(* IEC 61131-3 sources: Modbus-TCP-Traffic-Inspecting-via-OpenPLC-and-Wireshark/, 1 file *)

(* ---- program.st ---- *)
PROGRAM program0
  VAR
    Conveyor AT %QX100.0 : BOOL;
    Sensor AT %IX100.0 : BOOL;
  END_VAR

  Conveyor := Sensor;
END_PROGRAM

CONFIGURATION Config0

  RESOURCE Res0 ON PLC
    TASK task0(INTERVAL := T#20ms,PRIORITY := 0);
    PROGRAM instance0 WITH task0 : program0;
  END_RESOURCE
END_CONFIGURATION
